# EPICS autosave request: iocBoot/obsolete/ioc13xps_smkb/auto_settings.req
file "CARS_motor_settings.req",         P=$(P), M=m1
file "CARS_motor_settings.req",         P=$(P), M=m2
file "CARS_motor_settings.req",         P=$(P), M=m3
file "CARS_motor_settings.req",         P=$(P), M=m4
file "CARS_motor_settings.req",         P=$(P), M=m5
file "pseudoMotor_settings.req",        P=$(P), M=pm1
file "pseudoMotor_settings.req",        P=$(P), M=pm2
file "pseudoMotor_settings.req",        P=$(P), M=pm3
file "pseudoMotor_settings.req",        P=$(P), M=pm4
